{attribute addProperty BoxType "EL5102-0000-0016"}
{attribute addProperty Id "ControlAT %Q*Control_BA57B6F41621Set_counter_valueAT %Q*UDINT32417"}
{attribute addProperty CRC "3303417355"}
{attribute addProperty SizeInBites "48"}
{attribute addProperty SizeInBytes "6"}
TYPE ENC_Control_Channel_C4E6260B :
STRUCT
	{attribute addProperty Name "Control"}
	Control AT %Q* : Control_BA57B6F4;
	{attribute addProperty Name "Set_counter_value"}
	Set_counter_value AT %Q* : UDINT;
END_STRUCT
END_TYPE

(* stored: Version 1.2.0.0, ProductVersion 3.1.4024.9
   DUT ENC_Control_Channel_C4E6260B: Id {5b20f5d7-5ab5-4304-b672-61723f3fa79a} *)
